// TIA Portal V16 export
// export: Created 2021-08-30T10:49:30.03501Z, ExportSetting WithDefaults, DisplayName Totally Integrated Automation Portal, DisplayVersion V16 Update 3, DisplayName TIA Portal Version Control Interface, DisplayVersion V16 Update 2, DisplayName TIA Portal Openness, DisplayVersion V16 Update 3, DisplayName TIA Portal Teamcenter Gateway, DisplayVersion V16, DisplayName STEP 7 Professional, DisplayVersion V16 Update 3, DisplayName STEP 7 Safety, DisplayVersion V16, DisplayName WinCC Advanced, DisplayVersion V16 Update 3
FUNCTION_BLOCK "AllPID"   // FB3, FBD
{ S7_Optimized_Access := 'TRUE' }
VERSION : 0.1
// stored: AutoNumber true, IsIECCheckEnabled false, IsRetainMemResEnabled false, MemoryReserve 100, SetENOAutomatically false, UDAEnableTagReadback false
   VAR
      P30x { S7_SetPoint := 'True'} : "PID_Pump2Pu1Fc";
   END_VAR
BEGIN

REGION Network 1
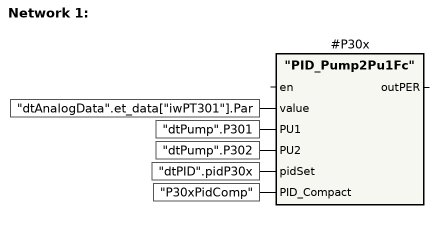
   #P30x(value := "dtAnalogData".et_data["iwPT301"].Par,   // "PID_Pump2Pu1Fc"
         PU1 := "dtPump".P301,
         PU2 := "dtPump".P302,
         pidSet := "dtPID".pidP30x,
         PID_Compact := "P30xPidComp");
END_REGION
END_FUNCTION_BLOCK
